{attribute 'linkalways'} 
{attribute 'no_explicit_call' := 'This FB is a CLASS and must be accessed using methods or properties'}
{attribute 'enable_dynamic_creation'}
FUNCTION_BLOCK FINAL NOT_LWORD EXTENDS Node
VAR
	in : _LWORD(0);
	out : _LWORD(0);
END_VAR

METHOD PUBLIC Clone : I_Node
VAR
	pNode : POINTER TO NOT_LWORD;
END_VAR
pNode := __NEW(NOT_LWORD);
Clone := pNode^;
END_METHOD

METHOD FB_init : BOOL
VAR_INPUT
	bInitRetains : BOOL; // if TRUE, the retain variables are initialized (warm start / cold start)
	bInCopyCode : BOOL;  // if TRUE, the instance afterwards gets moved into the copy code (online change)
END_VAR
AddInput('in',THIS^.in);
AddOutput('out', THIS^.out);
END_METHOD

METHOD PROTECTED OnExecute
VAR
END_VAR
out.Value := NOT in.Value;
END_METHOD

END_FUNCTION_BLOCK

(* stored: Version 1.1.0.1, ProductVersion 3.1.4024.15
   POU NOT_LWORD: Id {bfbab2ce-ece1-468d-a7ad-6aea56a4e7fe}, SpecialFunc None
   Folder Constructor: Id {72e660f8-f0ca-4bc9-a2ed-0c419eec973e}
   Method Clone: Id {cf45f9e1-6188-42ee-9406-d129986fc47d}
   Method FB_init: Id {e206ddde-6087-4ba6-bcda-7930a403fda0}
   Method OnExecute: Id {e4fb87e7-03ac-41af-8686-9aec33ebe919} *)
